Staubli VAL3: onF6Event.pgx

program onF6Event()
  local bool l_bYes
  local string l_sMessage
begin
  // look if the bButton is enable
  if bButton[5]
    //
  endIf
end
